// TIA Portal V20 export
// export: Created 2025-12-01T14:57:23.5502752Z, ExportSetting None, DisplayName Totally Integrated Automation Portal, DisplayVersion V20 Update 3, DisplayName TIA Portal Openness, DisplayVersion V20 Update 3, DisplayName TIA Portal Version Control Interface, DisplayVersion V20 Update 3, DisplayName STEP 7 Professional, DisplayVersion V20 Update 3, DisplayName STEP 7 Safety, DisplayVersion V20 Update 2, DisplayName WinCC Basic/Comfort/Advanced, DisplayVersion V20 Update 3, DisplayName WinCC Professional, DisplayVersion V20 Update 3, DisplayName WinCC Unified, DisplayVersion V20 Update 3
DATA_BLOCK "DB229_Listado_ordenes_sim"   // DB229
{ S7_Optimized_Access := 'TRUE' }
// stored: AutoNumber false, MemoryReserve 100
   VAR
      cruce : Array[1..500] of Struct
         orden : Array[1..50] of Byte;
      END_STRUCT;
   END_VAR
BEGIN
   cruce[1].orden[1] := 16#82;
   cruce[2].orden[1] := 16#80;
   cruce[3].orden[1] := 16#80;
   cruce[4].orden[1] := 16#80;
   cruce[10].orden[1..10] := 16#80;
   cruce[10].orden[11..12] := 16#00;
   cruce[16].orden[1] := 16#81;
   cruce[16].orden[2..4] := 16#00;
   cruce[16].orden[5..10] := 16#80;
   cruce[20].orden[1..10] := 16#80;
   cruce[45].orden[1..10] := 16#80;
END_DATA_BLOCK
